// TwinCAT 3 PLC project PLC
// ProgramVersion: 3.1.4024.12
// libraries:
//   Tc2_Standard, * (Beckhoff Automation GmbH)
//   Tc2_System, * (Beckhoff Automation GmbH)
//   Tc3_Module, * (Beckhoff Automation GmbH)
// project tree:
//   / PlcTask.TcTTO
//   POUs/ MAIN.TcPOU
// real-time tasks:
//   TASK PlcTask: cycle T#100000us, priority 20, ADS port 350

CONFIGURATION PLC
    RESOURCE PLC ON TwinCAT3
        TASK PlcTask(INTERVAL := T#100000us, PRIORITY := 20);
        PROGRAM MAIN WITH PlcTask : MAIN;
    END_RESOURCE
END_CONFIGURATION

// ---- POUs/MAIN.TcPOU
PROGRAM MAIN
VAR
	BoolTestVar    : BOOL;
	ByteTestVar    : BYTE;
	USIntTestVar   : USINT;
	SIntTestVar    : SINT;
	UIntTestVar    : UINT;
	WordTestVar    : WORD;
	UDIntTestVar   : UDINT;
	DWordTestVar   : DWORD;
	IntTestVar     : INT;
	DIntTestVar    : DINT;
	RealTestVar    : REAL;
	LRealTestVar   : LREAL;
	StringTestVar  : STRING;
	WStringTestVar : WSTRING;
	TimeTestVar    : TIME;
	DTTestVar      : DT;
	TODTestVar     : TOD;
	
	RNG              : DRAND;
	UIntChangingVar  : UINT;
	LRealChangingVar : LREAL;
END_VAR

BoolTestVar := TRUE;

ByteTestVar := 9;

USIntTestVar := 12;

SIntTestVar := -21;

UIntTestVar := 32;

WordTestVar := 54;

UDIntTestVar := 44;

DWordTestVar := 89;

IntTestVar := -23;

DIntTestVar := -23902;

RealTestVar := 2.03032;

LRealTestVar := -4.202902239210;

StringTestVar := WSTRING_TO_STRING("String test var value");

WStringTestVar := "WString test var value with extra ümlauts";

TimeTestVar := T#14MS;

DTTestVar := DT#1972-03-29-00:00:00;

TODTestVar := TOD#15:36:30.123;

RNG();
LRealChangingVar := LRealChangingVar + RNG.Num;

RNG();
UIntChangingVar := UIntChangingVar + LREAL_TO_UINT(RNG.Num);

END_PROGRAM
